// TIA Portal project "visualisation" (V17)

(* hardware
DEVICE "S7-1200 station_1"  S7-1200 Station
   slot 0: "Rack_0"  S7-1200 Rack  Rack  V1.0
   slot 1: "PLC_1"  CPU 1211C DC/DC/Rly  6ES7 211-1HE40-0XB0  V4.5
*)

// ===== PLC "PLC_1"  CPU 1211C DC/DC/Rly =====

VAR_GLOBAL   // PLC tag table "Default tag table"
   "System_Byte" AT %MB1 : Byte;
   "FirstScan" AT %M1.0 : Bool;
   "DiagStatusUpdate" AT %M1.1 : Bool;
   "AlwaysTRUE" AT %M1.2 : Bool;
   "AlwaysFALSE" AT %M1.3 : Bool;
   "Clock_Byte" AT %MB0 : Byte;
   "Clock_10Hz" AT %M0.0 : Bool;
   "Clock_5Hz" AT %M0.1 : Bool;
   "Clock_2.5Hz" AT %M0.2 : Bool;
   "Clock_2Hz" AT %M0.3 : Bool;
   "Clock_1.25Hz" AT %M0.4 : Bool;
   "Clock_1Hz" AT %M0.5 : Bool;
   "Clock_0.625Hz" AT %M0.6 : Bool;
   "Clock_0.5Hz" AT %M0.7 : Bool;
   "INT1" AT %MW2 : Int;
   "Tag_1" AT %M10.0 : Bool;
END_VAR

ORGANIZATION_BLOCK "Main"   // OB1, LAD, ProgramCycle
TITLE = "Main Program Sweep (Cycle)"
{ S7_Optimized_Access := 'TRUE' }
VERSION : 0.1
   VAR_INPUT
      Initial_Call : Bool;   // Initial call of this OB
      Remanence : Bool;   // =True, if remanent data are available
   END_VAR
   VAR_TEMP   // added for the SCL form of the ladder/FBD networks
      _w1 : Bool;
   END_VAR
BEGIN

REGION Network 1
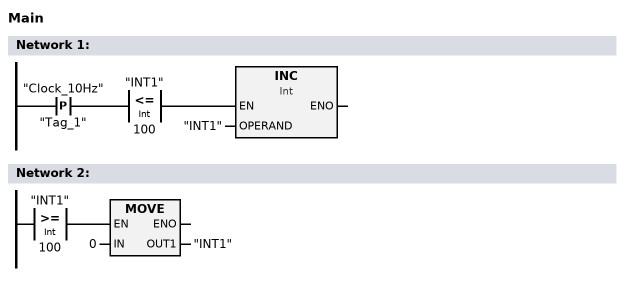
   RUNG wire#powerrail
      P_Contact(operand := "Clock_10Hz", bit := "Tag_1")
      { S7_Templates := "SrcType := Int" } LE_Contact(in1 := "INT1", in2 := 100)
      { S7_Templates := "DestType := Int" } Inc( "INT1" )
   END_RUNG
   // the same network as SCL:
   #_w1 := "Clock_10Hz" AND NOT "Tag_1";   // rising edge of "Clock_10Hz"
   "Tag_1" := "Clock_10Hz";
   IF #_w1 AND ("INT1" <= 100) THEN "INT1" := "INT1" + 1; END_IF;
END_REGION

REGION Network 2
   RUNG wire#powerrail
      { S7_Templates := "SrcType := Int" } GE_Contact(in1 := "INT1", in2 := 100)
      Move(in := 0, out1 => "INT1")
   END_RUNG
   // the same network as SCL:
   IF "INT1" >= 100 THEN "INT1" := 0; END_IF;
END_REGION
END_ORGANIZATION_BLOCK